FUNCTION_BLOCK Emitr
  (* Standard: 61499-2 *)
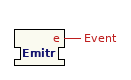
  EVENT_OUTPUT
    e;
  END_EVENT
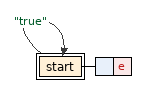
  EC_STATES
    start : -> e;
  END_STATES
  EC_TRANSITIONS
    start TO start := "true";
  END_TRANSITIONS
END_FUNCTION_BLOCK
